FUNCTION_BLOCK ILOCK_SWITCH_AX (* Prioritizes the last active input (Adapter Version). *)
  (* Standard: 61499-2; Description: Copyright (c) 2023 HR Agrartechnik GmbH This program and the accompanying materials are made available under the terms of the Eclipse Public License 2.0 which is available at https://www.eclipse.org/legal/epl-2.0/ SPDX-License-Identifier: EPL-2.0 *)
  (* Version 1.0, 2026-04-19, Franz Höpfinger, HR Agrartechnik GmbH, initial API and implementation and/or initial documentation *)
  PACKAGE logiBUS::signalprocessing::interlock;
  IMPORT eclipse4diac::core::TypeHash;
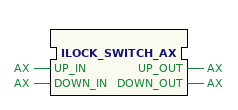
  SOCKETS
    UP_IN : adapter::types::unidirectional::AX; (* Input for forward/up direction *)
    DOWN_IN : adapter::types::unidirectional::AX; (* Input for backward/down direction *)
  END_SOCKETS
  PLUGS
    UP_OUT : adapter::types::unidirectional::AX; (* Output for forward/up direction *)
    DOWN_OUT : adapter::types::unidirectional::AX; (* Output for backward/down direction *)
  END_PLUGS
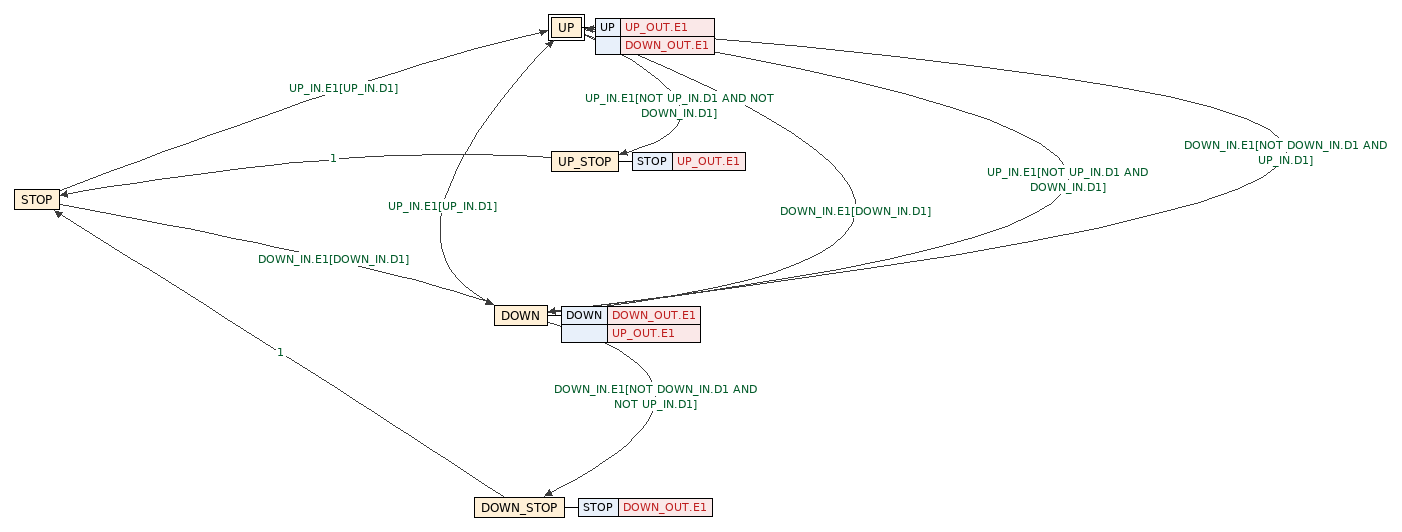
  EC_STATES
    UP : UP -> UP_OUT.E1, -> DOWN_OUT.E1;
    DOWN : DOWN -> DOWN_OUT.E1, -> UP_OUT.E1;
    STOP;
    UP_STOP : STOP -> UP_OUT.E1;
    DOWN_STOP : STOP -> DOWN_OUT.E1;
  END_STATES
  EC_TRANSITIONS
    STOP TO UP := UP_IN.E1[UP_IN.D1];
    STOP TO DOWN := DOWN_IN.E1[DOWN_IN.D1];
    UP TO DOWN := DOWN_IN.E1[DOWN_IN.D1];
    UP TO DOWN := UP_IN.E1[NOT UP_IN.D1 AND DOWN_IN.D1];
    UP TO UP_STOP := UP_IN.E1[NOT UP_IN.D1 AND NOT DOWN_IN.D1];
    DOWN TO UP := UP_IN.E1[UP_IN.D1];
    DOWN TO UP := DOWN_IN.E1[NOT DOWN_IN.D1 AND UP_IN.D1];
    DOWN TO DOWN_STOP := DOWN_IN.E1[NOT DOWN_IN.D1 AND NOT UP_IN.D1];
    UP_STOP TO STOP := 1;
    DOWN_STOP TO STOP := 1;
  END_TRANSITIONS
  ALGORITHM UP IN ST:
UP_OUT.D1 := BOOL#TRUE;
DOWN_OUT.D1 := BOOL#FALSE;
  END_ALGORITHM
  ALGORITHM DOWN IN ST:
UP_OUT.D1 := BOOL#FALSE;
DOWN_OUT.D1 := BOOL#TRUE;
  END_ALGORITHM
  ALGORITHM STOP IN ST:
UP_OUT.D1 := BOOL#FALSE;
DOWN_OUT.D1 := BOOL#FALSE;
  END_ALGORITHM
END_FUNCTION_BLOCK
